Fanuc KAREL source: PROG_CLEAR.kl

PROGRAM T
%NOLOCKGROUP
VAR
 v0 : STRING[40]
 v1 : INTEGER
 v2 : INTEGER
BEGIN
 PROG_CLEAR(v0, v1, v2)
END T
